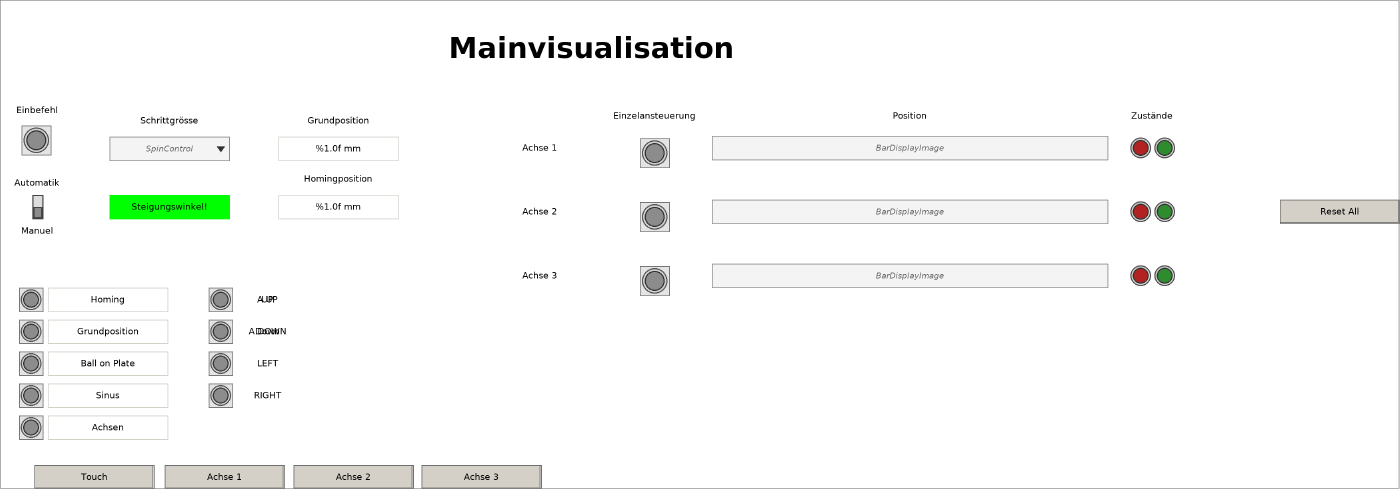
VISUALIZATION Mainvisu  // 1750x612
    DipSwitch (32,244 31x30), variable: GVL.Automatik, behaviour: TOGGLE, style: Switch-DipSwitch-Gray
    Label (12,214 69x30), "Automatik"
    Label (12,274 69x30), "Manuel"
    PushSwitch (260,360 32x30), variable: GVL.UP, invisible if: GVL.Achsenkontrolle, behaviour: TAP, style: Switch-PushSwitch-Gray
    PushSwitch (260,400 32x30), variable: GVL.Down, invisible if: GVL.Achsenkontrolle, behaviour: TAP, style: Switch-PushSwitch-Gray
    Label (300,360 69x30), "UP", invisible if: GVL.Achsenkontrolle
    Label (300,400 69x30), "Down", invisible if: GVL.Achsenkontrolle
    Label (348,136 150x30), "Grundposition"
    PushSwitch (22,400 34x30), variable: GVL.Grundposition, behaviour: TAP, style: Switch-PushSwitch-Gray
    Textfield (348,171 150x30), "%1.0f mm", text variable: GVL.Eingabe_Sollposition
    Label (348,209 150x30), "Homingposition"
    Textfield (348,244 150x30), "%1.0f mm", text variable: GVL.Eingabe_Grundposition
    Label (12,123 69x30), "Einbefehl"
    SpinControl (137,171 150x30), variable: GVL.n
    Label (137,136 150x30), "Schrittgrösse"
    BarDisplayImage (890,170 495x30), value: MAIN.Axis_R.ActualPosition, style: BarDisplayImage-Gray, scale format: %.0f, scale 0..200
    Label (890,130 495x30), "Position"
    BarDisplayImage (890,250 495x30), value: MAIN.Axis_S.ActualPosition, style: BarDisplayImage-Gray, scale format: %.0f, scale 0..200
    BarDisplayImage (890,330 495x30), value: MAIN.Axis_T.ActualPosition, style: BarDisplayImage-Gray, scale format: %.0f, scale 0..200
    Lamp1 (1410,170 32x30), variable: MAIN.Axis_R.WarningActive, style: Lamp-Lamp1-Red
    Lamp1 (1410,250 32x30), variable: MAIN.Axis_S.WarningActive, style: Lamp-Lamp1-Red
    Lamp1 (1410,330 32x30), variable: MAIN.Axis_T.WarningActive, style: Lamp-Lamp1-Red
    Lamp1 (1440,170 32x30), variable: MAIN.Axis_R.Ready, style: Lamp-Lamp1-Green
    Lamp1 (1440,250 32x30), variable: MAIN.Axis_S.Ready, style: Lamp-Lamp1-Green
    Lamp1 (1440,330 32x30), variable: MAIN.Axis_T.Ready, style: Lamp-Lamp1-Green
    PushSwitchLed (800,170 37x43), variable: MAIN.Axis_R.bManual, behaviour: TOGGLE, style: Switch-PushSwitchLed-Gray
    PushSwitchLed (800,250 37x43), variable: MAIN.Axis_S.bManual, behaviour: TOGGLE, style: Switch-PushSwitchLed-Gray
    PushSwitchLed (800,330 37x43), variable: MAIN.Axis_T.bManual, behaviour: TOGGLE, style: Switch-PushSwitchLed-Gray
    Label (743,130 150x30), "Einzelansteuerung"
    PushSwitchLed (27,154 37x43), variable: gvl.V48VDC_Einbefehl, behaviour: TOGGLE, style: Switch-PushSwitchLed-Gray
    PushSwitch (22,440 34x30), variable: GVL.BndP, behaviour: TAP, style: Switch-PushSwitch-Gray
    Textfield (60,440 150x30), "Ball on Plate", colour toggle: GVL.BNP_Aktiv
        toggle GVL.BndP
    PushSwitch (22,480 34x30), variable: GVL.Sinus, behaviour: TAP, style: Switch-PushSwitch-Gray
    Textfield (60,480 150x30), "Sinus", colour toggle: GVL.Sinus_Aktiv
        toggle GVL.BndP
    Textfield (60,400 150x30), "Grundposition", colour toggle: GVL.Position_Aktiv
        toggle GVL.BndP
    Textfield (137,244 150x30), "Steigungswinkel!", colour toggle: GVL.Warnung_Steigungswinkel
        toggle GVL.BndP
    PushSwitch (260,360 32x30), variable: GVL.XAchseUp, invisible if: not GVL.Achsenkontrolle, behaviour: TAP, style: Switch-PushSwitch-Gray
    PushSwitch (260,400 32x30), variable: GVL.XAchseDown, invisible if: not GVL.Achsenkontrolle, behaviour: TAP, style: Switch-PushSwitch-Gray
    Label (300,360 69x30), "A UP", invisible if: not GVL.Achsenkontrolle
    Label (300,400 69x30), "A DOWN", invisible if: not GVL.Achsenkontrolle
    PushSwitch (260,440 32x30), variable: GVL.YAchseDown, invisible if: not GVL.Achsenkontrolle, behaviour: TAP, style: Switch-PushSwitch-Gray
    PushSwitch (260,480 32x30), variable: GVL.YAchseUp, invisible if: not GVL.Achsenkontrolle, behaviour: TAP, style: Switch-PushSwitch-Gray
    Label (300,440 69x30), "LEFT", invisible if: not GVL.Achsenkontrolle
    Label (300,480 69x30), "RIGHT", invisible if: not GVL.Achsenkontrolle
    Textfield (60,520 150x30), "Achsen", colour toggle: GVL.Achsenkontrolle
    PushSwitch (22,360 34x30), variable: GVL.Homing, behaviour: TAP, style: Switch-PushSwitch-Gray
    Textfield (60,360 150x30), "Homing", colour toggle: GVL.eingabesperre
        toggle GVL.BndP
    PushSwitch (22,520 34x30), variable: GVL.AchsenkontrolleVisu, behaviour: TAP, style: Switch-PushSwitch-Gray
    Label (600,170 150x30), "Achse 1"
    Label (600,250 150x30), "Achse 2"
    Label (600,330 150x30), "Achse 3"
    Label (1410,130 60x30), "Zustände"
    Label (3,4 1473x112), "Mainvisualisation"
    Button (206,582 150x30), "Achse 1"
        OnMouseDown: change screen: Achse_R
    Button (43,582 150x30), "Touch"
        OnMouseDown: change screen: Touch
    Button (367,582 150x30), "Achse 2"
        OnMouseDown: change screen: Achse_S
    Button (527,582 150x30), "Achse 3"
        OnMouseDown: change screen: Achse_T
    Button (1600,250 150x30), "Reset All"
        tap GVL.reset
END_VISUALIZATION

(* stored: Version 1.1.0.1, ProductVersion 3.1.4024.10
   Visu Mainvisu: Id {2f2efe17-56e7-4248-bc9f-434a0baf1bfb} *)
